{attribute 'linkalways'} 
{attribute 'no_explicit_call' := 'This FB is a CLASS and must be accessed using methods or properties'}
{attribute 'enable_dynamic_creation'}
FUNCTION_BLOCK FINAL MOD_UINT EXTENDS Node
VAR
	in1 : _UINT(0);
	in2 : _UINT(0);
	out : _UINT(0);
END_VAR

METHOD PUBLIC Clone : I_Node
VAR
	pNode : POINTER TO MOD_UINT;
END_VAR
pNode := __NEW(MOD_UINT);
Clone := pNode^;
END_METHOD

METHOD FB_init : BOOL
VAR_INPUT
	bInitRetains : BOOL; // if TRUE, the retain variables are initialized (warm start / cold start)
	bInCopyCode : BOOL;  // if TRUE, the instance afterwards gets moved into the copy code (online change)
END_VAR
AddInput('in1',THIS^.in1);
AddInput('in2',THIS^.in2);
AddOutput('out', THIS^.out);
END_METHOD

METHOD PROTECTED OnExecute
VAR
END_VAR
out.Value := in1.Value MOD in2.Value;
END_METHOD

END_FUNCTION_BLOCK

(* stored: Version 1.1.0.1, ProductVersion 3.1.4024.15
   POU MOD_UINT: Id {abf4dd9b-dd10-4200-875a-52cdc0464c0d}, SpecialFunc None
   Folder Constructor: Id {1e433081-0d7d-4be5-9861-62ca7bd962f4}
   Method Clone: Id {63a1875a-0b74-4c45-986a-044ef043d754}
   Method FB_init: Id {9fd86127-c34c-4880-8958-993066b7e246}
   Method OnExecute: Id {6bef5de6-c7b5-405b-adb5-d6f4af1fe91c} *)
